(*
Casts I_Component as I_Signal.
Returns:
- Ok - Success,
- Err.InvRef - Invalid reference,
- Err.Itf0 - Invalid interface,
- Err.NoMatch - Cast failed
*)
FUNCTION ICompToISignal : Result
VAR_INPUT
	iIn	: I_Component;
	iOut: REFERENCE TO I_Signal;
END_VAR

IF NOT __ISVALIDREF(iOut) THEN
	ICompToISignal := Err.InvRef;
	RETURN;
END_IF

IF iIn = 0 THEN
	ICompToISignal := Err.Itf0;
	RETURN;
END_IF

IF __QUERYINTERFACE(iIn, iOut) THEN
	ICompToISignal := Ok;
ELSE
	ICompToISignal := Err.NoMatch;
END_IF

END_FUNCTION

(* stored: Version 1.1.0.1
   POU ICompToISignal: Id {5f959340-f887-4136-afe4-e25a563d68c5}, SpecialFunc None *)
